{attribute 'qualified_only'}
VAR_GLOBAL CONSTANT PERSISTENT
	NUMBER_ALARMS : UINT := 1;
END_VAR

(* stored: Version 1.1.0.1, ProductVersion 3.1.4024.12
   GVL IonizerConst: Id {48a480e9-e246-4ca3-9361-828a37c4da0b}, ParameterList True *)
